TYPE STATE:
    STRUCT
        curTime: REAL;
        dvar_M_p_vt: BOOL;
        dvar_M_p_vf: BOOL;
        dvar_M_p_vr2: DINT;
        dvar_M_p_vr3: DINT;
        dvar_M_p_v0: DINT;
        dvar_M_p_v1: DINT;
        dvar_M_p_v2: DINT;
        dvar_M_p_v3: DINT;
        dvar_M_p_v123: DINT;
        dvar_M_p_vn1: DINT;
        dvar_M_p_vn2: DINT;
        dvar_M_p_v00: REAL;
        dvar_M_p_v01: REAL;
        dvar_M_p_v05: REAL;
        dvar_M_p_v10: REAL;
        dvar_M_p_v20: REAL;
        dvar_M_p_v30: REAL;
        dvar_M_p_v270: REAL;
        dvar_M_p_vn01: REAL;
        dvar_M_p_vn10: REAL;
        dvar_M_p_e: REAL;
        dvar_M_p_ve1: DINT;
        dvar_M_p_ve2: DINT;
        dvar_M_p_ve3: DINT;
        dvar_M_p_ve4: DINT;
        dvar_M_p_vbir: TupleStruct_2;
        dvar_M_p_vb000: BOOL;
        dvar_M_p_vb001: BOOL;
        dvar_M_p_vb002: BOOL;
        dvar_M_p_vb003: BOOL;
        dvar_M_p_vb004: BOOL;
        dvar_M_p_vb005: BOOL;
        dvar_M_p_vb006: BOOL;
        dvar_M_p_vb007: BOOL;
        dvar_M_p_vb008: BOOL;
        dvar_M_p_vb009: BOOL;
        dvar_M_p_vb010: BOOL;
        dvar_M_p_vb011: BOOL;
        dvar_M_p_vb012: BOOL;
        dvar_M_p_vb013: BOOL;
        dvar_M_p_vb014: BOOL;
        dvar_M_p_vb015: BOOL;
        dvar_M_p_vb016: BOOL;
        dvar_M_p_vb017: BOOL;
        dvar_M_p_vb018: BOOL;
        dvar_M_p_vb019: BOOL;
        dvar_M_p_vb020: BOOL;
        dvar_M_p_vb021: BOOL;
        dvar_M_p_vb022: BOOL;
        dvar_M_p_vb023: BOOL;
        dvar_M_p_vb024: BOOL;
        dvar_M_p_vb025: BOOL;
        dvar_M_p_vb026: BOOL;
        dvar_M_p_vb027: BOOL;
        dvar_M_p_vb028: BOOL;
        dvar_M_p_vb029: BOOL;
        dvar_M_p_vb030: BOOL;
        dvar_M_p_vb031: BOOL;
        dvar_M_p_vb032: BOOL;
        dvar_M_p_vb033: BOOL;
        dvar_M_p_vb034: BOOL;
        dvar_M_p_vb035: BOOL;
        dvar_M_p_vb036: BOOL;
        dvar_M_p_vb037: BOOL;
        dvar_M_p_vb038: BOOL;
        dvar_M_p_vb039: BOOL;
        dvar_M_p_vb040: BOOL;
        dvar_M_p_vb041: BOOL;
        dvar_M_p_vb042: BOOL;
        dvar_M_p_vb043: BOOL;
        dvar_M_p_vb044: BOOL;
        dvar_M_p_vb045: BOOL;
        dvar_M_p_vb046: BOOL;
        dvar_M_p_vb047: BOOL;
        dvar_M_p_vb048: BOOL;
        dvar_M_p_vb049: BOOL;
        dvar_M_p_vb050: BOOL;
        dvar_M_p_vb051: BOOL;
        dvar_M_p_vb052: BOOL;
        dvar_M_p_vb053: BOOL;
        dvar_M_p_vb054: BOOL;
        dvar_M_p_vb055: BOOL;
        dvar_M_p_vb056: BOOL;
        dvar_M_p_vb057: BOOL;
        dvar_M_p_vb058: BOOL;
        dvar_M_p_vb059: BOOL;
        dvar_M_p_vb060: BOOL;
        dvar_M_p_vb061: BOOL;
        dvar_M_p_vb062: BOOL;
        dvar_M_p_vb063: BOOL;
        dvar_M_p_vb064: BOOL;
        dvar_M_p_vb065: BOOL;
        dvar_M_p_vb066: BOOL;
        dvar_M_p_vb067: BOOL;
        dvar_M_p_vb068: BOOL;
        dvar_M_p_vb069: BOOL;
        dvar_M_p_vb070: BOOL;
        dvar_M_p_vb071: BOOL;
        dvar_M_p_vb072: BOOL;
        dvar_M_p_vb073: BOOL;
        dvar_M_p_vb074: BOOL;
        dvar_M_p_vb075: BOOL;
        dvar_M_p_vb076: BOOL;
        dvar_M_p_vb077: BOOL;
        dvar_M_p_vb078: BOOL;
        dvar_M_p_vb079: BOOL;
        dvar_M_p_vb080: BOOL;
        dvar_M_p_vb081: BOOL;
        dvar_M_p_vb082: BOOL;
        dvar_M_p_vb083: BOOL;
        dvar_M_p_vb084: BOOL;
        dvar_M_p_vb085: BOOL;
        dvar_M_p_vb086: BOOL;
        dvar_M_p_vb087: BOOL;
        dvar_M_p_vb088: BOOL;
        dvar_M_p_vb089: BOOL;
        dvar_M_p_vb090: BOOL;
        dvar_M_p_vb091: BOOL;
        dvar_M_p_vb092: BOOL;
        dvar_M_p_vb093: BOOL;
        dvar_M_p_vb094: BOOL;
        dvar_M_p_vb095: BOOL;
        dvar_M_p_vb096: BOOL;
        dvar_M_p_vb097: BOOL;
        dvar_M_p_vb098: BOOL;
        dvar_M_p_vb099: BOOL;
        dvar_M_p_vi00: DINT;
        dvar_M_p_vi01: DINT;
        dvar_M_p_vi02: DINT;
        dvar_M_p_vi03: DINT;
        dvar_M_p_vi04: DINT;
        dvar_M_p_vi05: DINT;
        dvar_M_p_vi06: DINT;
        dvar_M_p_vi07: DINT;
        dvar_M_p_vi08: DINT;
        dvar_M_p_vi09: DINT;
        dvar_M_p_vi10: DINT;
        dvar_M_p_vi11: DINT;
        dvar_M_p_vi12: DINT;
        dvar_M_p_vi13: DINT;
        dvar_M_p_vi14: DINT;
        dvar_M_p_vi15: DINT;
        dvar_M_p_vi16: DINT;
        dvar_M_p_vi17: DINT;
        dvar_M_p_vi18: DINT;
        dvar_M_p_vi19: DINT;
        dvar_M_p_vi20: DINT;
        dvar_M_p_vi21: DINT;
        dvar_M_p_vi22: DINT;
        dvar_M_p_vi23: DINT;
        dvar_M_p_vi24: DINT;
        dvar_M_p_vi25: DINT;
        dvar_M_p_vi26: DINT;
        dvar_M_p_vi27: DINT;
        dvar_M_p_vi28: DINT;
        dvar_M_p_vi29: DINT;
        dvar_M_p_vi30: DINT;
        dvar_M_p_vi31: DINT;
        dvar_M_p_vi32: DINT;
        dvar_M_p_vi33: DINT;
        dvar_M_p_vi34: DINT;
        dvar_M_p_vr00: REAL;
        dvar_M_p_vr01: REAL;
        dvar_M_p_vr02: REAL;
        dvar_M_p_vr03: REAL;
        dvar_M_p_vr04: REAL;
        dvar_M_p_vr05: REAL;
        dvar_M_p_vr06: REAL;
        dvar_M_p_vr07: REAL;
        dvar_M_p_vr08: REAL;
        dvar_M_p_vr09: REAL;
        dvar_M_p_vr10: REAL;
        dvar_M_p_vr11: REAL;
        dvar_M_p_vr12: REAL;
        dvar_M_p_vr13: REAL;
        dvar_M_p_vr14: REAL;
        dvar_M_p_vr15: REAL;
        dvar_M_p_vr16: REAL;
        dvar_M_p_vr17: REAL;
        dvar_M_p_vr18: REAL;
        dvar_M_p_vr19: REAL;
        dvar_M_p_vr20: REAL;
        dvar_M_p_vr21: REAL;
        dvar_M_p_vr22: REAL;
        dvar_M_p_vr23: REAL;
        dvar_M_p_vr24: REAL;
        dvar_M_p_vr25: REAL;
        dvar_M_p_vr26: REAL;
        dvar_M_p_vr27: REAL;
        dvar_M_p_vr28: REAL;
        dvar_M_p_vr29: REAL;
        dvar_M_p_vr30: REAL;
        dvar_M_p_vr31: REAL;
        dvar_M_p_vr32: REAL;
        dvar_M_p_vr33: REAL;
        dvar_M_p_vr34: REAL;
        dvar_M_p_vr35: REAL;
        dvar_M_p_vr36: REAL;
        dvar_M_p_vr37: REAL;
        dvar_M_p_vr38: REAL;
        dvar_M_p_vr39: REAL;
        dvar_M_p_vr40: REAL;
        dvar_M_p_vr41: REAL;
        dvar_M_p_vr42: REAL;
        dvar_M_p_vr43: REAL;
        dvar_M_p_vr44: REAL;
        dvar_M_p_vr45: REAL;
        dvar_M_p_vr46: REAL;
        dvar_M_p_vr47: REAL;
        dvar_M_p_vr48: REAL;
        dvar_M_p_vr49: REAL;
        dvar_M_p_vr50: REAL;
        dvar_M_p_vr51: REAL;
        dvar_M_p_vr52: REAL;
        dvar_M_p_vr53: REAL;
        dvar_M_p_vr54: REAL;
        dvar_M_p_vr55: REAL;
        dvar_M_p_vr56: REAL;
        dvar_M_p_vr57: REAL;
        dvar_M_p_vr58: REAL;
        dvar_M_p: DINT;
    END_STRUCT;
END_TYPE
